(* Logix 5000 project; controller ACDTests 1756-L85E rev 34.11; software revision 34.01 *)
// Controller Description

TASK MainTask (continuous, watchdog 500 ms) : MainProgram

MODULES
   Local : 1756-L85E (ICP 0, rev 34.11)
      ETH_MODULE : 1756-EN2T (ICP 1, Ethernet 192.168.1.2, rev 11.1)   // ETH_MODULE Description
END_MODULES

ADD_ON_INSTRUCTION AddOnInstruction   (* revision 1.7 ExtendedText, vendor ACD-TOOLS *)
// AddOnInstruction Description
// Revision note:
// Revision Note Add On Instruction
VAR
   AOIDINTLocalTag : DINT := 666; {access None}   // AOILocalTagDescription
END_VAR

ROUTINE Logic   (* ladder *)
   0: NOP();
END_ROUTINE
END_ADD_ON_INSTRUCTION

VAR_GLOBAL   (* controller tags *)
   a5000_String32 : AB:5000_String32_Struct:I:0;
   AliasTag5000String32 : ALIAS FOR a5000_String32.LEN;
   Constant : DINT; {constant}
   DATETIME_RadixDateTime : DT;
   DINT : DINT;   // DINT_DESCRIPTION
   INT : INT;   // INT Description
   LDATETIME_RadixNanoSec : LDT;
   LTIME_RadixLTime : LTIME;
   NoAccess : DINT; {access None}
   RadixASCII : DINT;
   RadixBinary : DINT;
   RadixExponential : REAL;
   RadixFloat : REAL;
   RadixHex : DINT;
   RadixOctal : DINT;
   ReadOnly : DINT; {access Read Only}
   TIME32_RadixTime32 : TIME32;
   TIME_RadixTimeUs : TIME;
   UDINT : UDINT;   // UDINT Description
   UINT : UINT;   // UINT Description
   ULINT : ULINT;   // ULINT Description
END_VAR

PROGRAM MainProgram   (* main routine MainRoutine *)
VAR
   AND_01 : FBD_LOGICAL;
   BAND_01 : FBD_BOOLEAN_AND := (In1 := 1, In2 := 1, In3 := 1, In4 := 1, In5 := 1, In6 := 1, In7 := 1, In8 := 1);
   BOR_01 : FBD_BOOLEAN_OR;
   MainProgramLocalTag : DINT;   // MainProgramLocalTagDescription
   MainProgramLocalTagNoAccess : DINT; {access None}   // MainProgramLocalTagDescription
   MainProgramLocalTagReadOnly : DINT; {access Read Only}   // MainProgramLocalTagDescription
   Step_000 : SFC_STEP := (Status := 16#0020_0000, PauseTimer := 1);
   Stop_000 : SFC_STOP;
   Tran_000 : BOOL;
END_VAR
VAR_INPUT
   MainProgramInputParameter : DINT;
END_VAR
VAR_OUTPUT
   MainProgramOutputParameter : DINT; {access Read Only}
END_VAR
VAR {public}
   MainProgramPublicParameters : DINT;
END_VAR

ROUTINE FBDRoutine   (* function block diagram *)
// FBDRoutineDescription
   SHEET 1
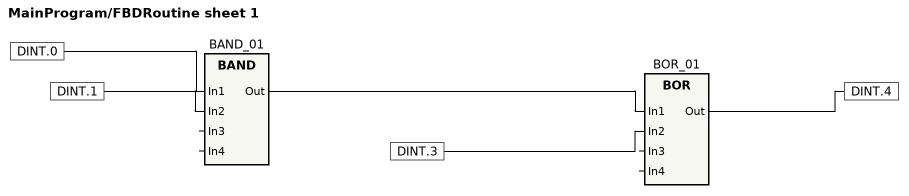
   BAND_01 : BAND(In1 := DINT.0, In2 := DINT.1);   // unwired pins: In3 In4
   BOR_01 : BOR(In1 := BAND_01.Out, In2 := DINT.3);   // unwired pins: In3 In4
   DINT.4 := BOR_01.Out;
   SHEET 2
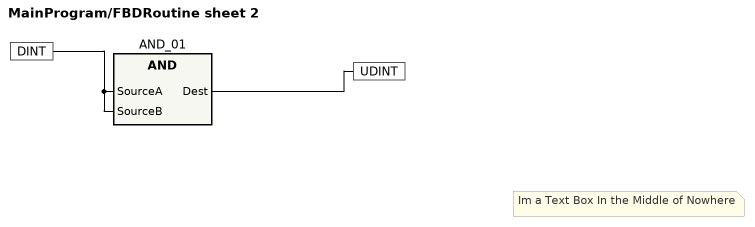
   // Im a Text Box In the Middle of Nowhere
   AND_01 : AND(SourceA := DINT, SourceB := DINT);
   UDINT := AND_01.Dest;
END_ROUTINE

ROUTINE MainRoutine   (* ladder *)
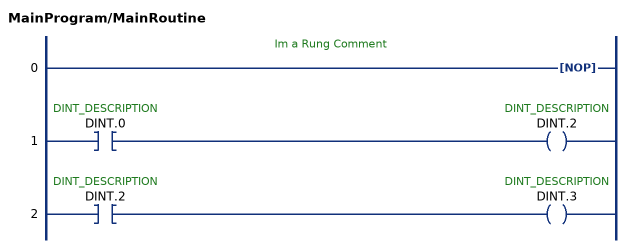
   // Im a Rung Comment
   0: NOP();
   1: XIC(DINT.0)OTE(DINT.2);
   2: XIC(DINT.2)OTE(DINT.3);
END_ROUTINE

ROUTINE SequentialFunctionChart   (* sequential function chart *)
// SequenceFunctionChartRoutineDescription
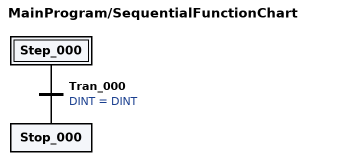
   INITIAL_STEP Step_000:
   END_STEP
   TRANSITION Tran_000 FROM Step_000 TO Stop_000
      := DINT = DINT
   END_TRANSITION
   STOP Stop_000;
END_ROUTINE

ROUTINE STRoutine   (* structured text *)
// STRoutineDescrioption
   DINT := DINT AND UDINT; // Line 1 COmment
   DINT := DINT AND ULINT; // Line 2 Comment
   
   // Random Comment
   
   
END_ROUTINE
END_PROGRAM
